// TIA Portal V20 export
// export: Created 2025-12-01T14:57:43.6224422Z, ExportSetting None, DisplayName Totally Integrated Automation Portal, DisplayVersion V20 Update 3, DisplayName TIA Portal Openness, DisplayVersion V20 Update 3, DisplayName TIA Portal Version Control Interface, DisplayVersion V20 Update 3, DisplayName STEP 7 Professional, DisplayVersion V20 Update 3, DisplayName STEP 7 Safety, DisplayVersion V20 Update 2, DisplayName WinCC Basic/Comfort/Advanced, DisplayVersion V20 Update 3, DisplayName WinCC Professional, DisplayVersion V20 Update 3, DisplayName WinCC Unified, DisplayVersion V20 Update 3
FUNCTION "FC509_SIM_Ordenes_SRC_Clasificador_V2" : Void   // FC509, LAD
{ S7_Optimized_Access := 'FALSE' }
AUTHOR : ROUTER
NAME : 20190911
VERSION : 3.1
// NIEVES: 2024/01/29
// Para que en los cruces de más de un destino sea más facil configurar cuantas cajas enviamos por cada cruce, y además hacerlo de la manera más simple para los cruces configurados de manera especial, se configuran en un db las ordenes que queremos que se vayan extrayendo, de manera que podremos decidir en cada momento cuantas enviamos por cada desvío, y la orden que necesitamos para que se ejecute correctamente.
// stored: AutoNumber false, SetENOAutomatically false
   VAR_INPUT
      Numero_cruce : UInt;
      Sacar_orden : Bool;
      Reset : Bool;
   END_VAR
   VAR_OUTPUT
      Orden_FIFO : "ROUT_Orden_Fifo_Scanner";
   END_VAR
   VAR_IN_OUT
      Mem_FP : Bool;
      Aux_contador_cajas : UDInt;
   END_VAR
   VAR_TEMP
      aux_SSCC : DInt;
   END_VAR
   VAR_TEMP   // added for the SCL form of the ladder/FBD networks
      _w1 : Bool;
      _w2 : Bool;
   END_VAR
BEGIN

REGION Network 1: inicializacion
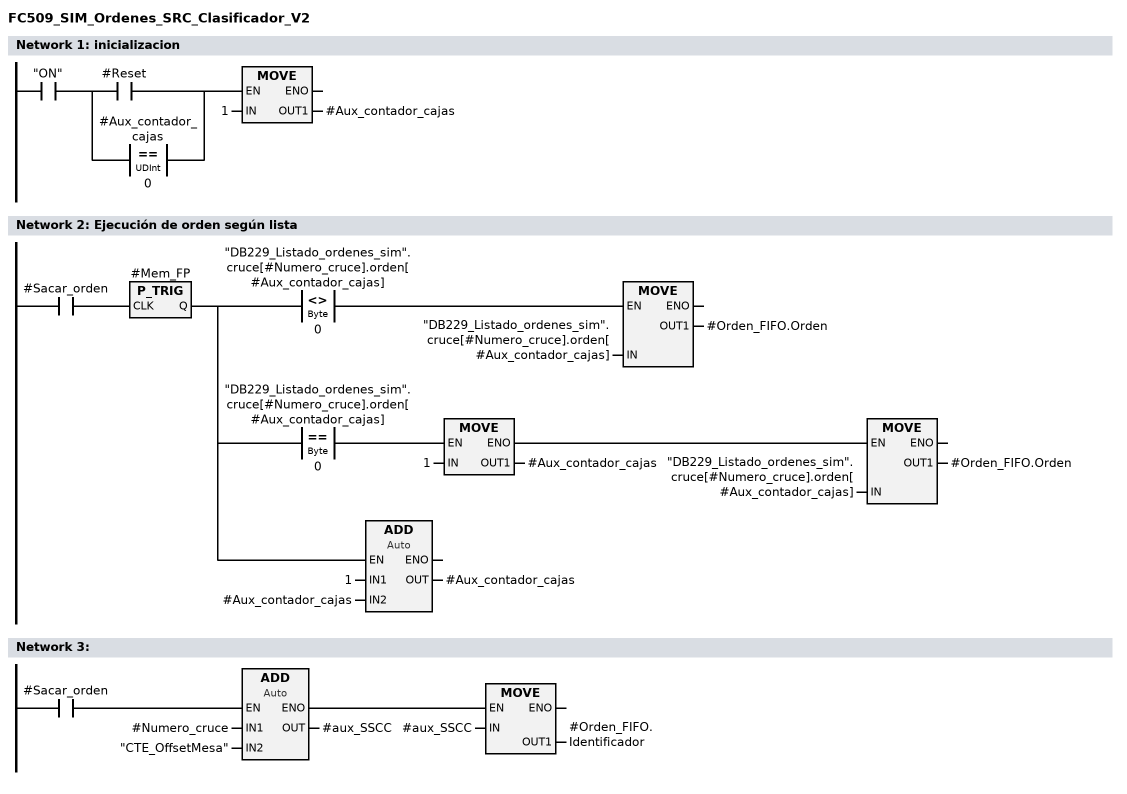
   RUNG wire#powerrail
      Contact( "ON" )
      wire#w1
      Contact( #Reset )
      wire#w2
      Move(in := 1, out1 => #Aux_contador_cajas)
   END_RUNG
   RUNG wire#w1
      { S7_Templates := "SrcType := UDInt" } EQ_Contact(in1 := #Aux_contador_cajas, in2 := 0)
   END_RUNG wire#w2
   // the same network as SCL:
   IF "ON" AND (#Reset OR (#Aux_contador_cajas = 0)) THEN #Aux_contador_cajas := 1; END_IF;
END_REGION

REGION Network 2: Ejecución de orden según lista
   RUNG wire#powerrail
      Contact( #Sacar_orden )
      P_Trig( #Mem_FP )
      wire#w1
      { S7_Templates := "SrcType := Byte" } NE_Contact(in1 := "DB229_Listado_ordenes_sim".cruce[#Numero_cruce].orden[#Aux_contador_cajas], in2 := 0)
      Move(in := "DB229_Listado_ordenes_sim".cruce[#Numero_cruce].orden[#Aux_contador_cajas], out1 => #Orden_FIFO.Orden)
   END_RUNG
   RUNG wire#w1
      { S7_Templates := "SrcType := Byte" } EQ_Contact(in1 := "DB229_Listado_ordenes_sim".cruce[#Numero_cruce].orden[#Aux_contador_cajas], in2 := 0)
      Move(in := 1, out1 => #Aux_contador_cajas)
      Move(in := "DB229_Listado_ordenes_sim".cruce[#Numero_cruce].orden[#Aux_contador_cajas], out1 => #Orden_FIFO.Orden)
   END_RUNG
   RUNG wire#w1
      Add(in1 := 1, in2 := #Aux_contador_cajas, out => #Aux_contador_cajas)
   END_RUNG
   // the same network as SCL:
   #_w1 := #Sacar_orden AND NOT #Mem_FP;   // rising edge
   #Mem_FP := #Sacar_orden;
   IF #_w1 AND ("DB229_Listado_ordenes_sim".cruce[#Numero_cruce].orden[#Aux_contador_cajas] <> 0) THEN
       #Orden_FIFO.Orden := "DB229_Listado_ordenes_sim".cruce[#Numero_cruce].orden[#Aux_contador_cajas];
   END_IF;
   #_w2 := #_w1 AND ("DB229_Listado_ordenes_sim".cruce[#Numero_cruce].orden[#Aux_contador_cajas] = 0);
   IF #_w2 THEN
       #Aux_contador_cajas := 1;
       #Orden_FIFO.Orden := "DB229_Listado_ordenes_sim".cruce[#Numero_cruce].orden[#Aux_contador_cajas];
   END_IF;
   IF #_w1 THEN #Aux_contador_cajas := 1 + #Aux_contador_cajas; END_IF;
END_REGION

REGION Network 3
   RUNG wire#powerrail
      Contact( #Sacar_orden )
      Add(in1 := #Numero_cruce, in2 := "CTE_OffsetMesa", out => #aux_SSCC)
      Move(in := #aux_SSCC, out1 => #Orden_FIFO.Identificador)
   END_RUNG
   // the same network as SCL:
   IF #Sacar_orden THEN
       #aux_SSCC := #Numero_cruce + "CTE_OffsetMesa";
       #Orden_FIFO.Identificador := #aux_SSCC;
   END_IF;
END_REGION
END_FUNCTION
